// TIA Portal V20 export
FUNCTION_BLOCK "Conveyor_C2"   // FB3, FBD
// stored: Access Published, MemoryReserve 100, Namespace Conveyor2, SetENOAutomatically false
   VAR
      Jog_Right : Bool;
      Jog_Left : Bool;
      Auto_Right : Bool;
      PF_Bay1_NewProd : Bool;
      PF_Bay2_NewProd : Bool;
      PF_Bay3_NewProd : Bool;
      PF_Bay4_EndConv : Bool;
   END_VAR
   VAR_TEMP   // added for the SCL form of the ladder/FBD networks
      _w1 : Bool;
      _w2 : Bool;
      _w3 : Bool;
      _w4 : Bool;
      _w5 : Bool;
      _w6 : Bool;
      _w7 : Bool;
   END_VAR
BEGIN

REGION Network 1: Jog conveyor LEFT
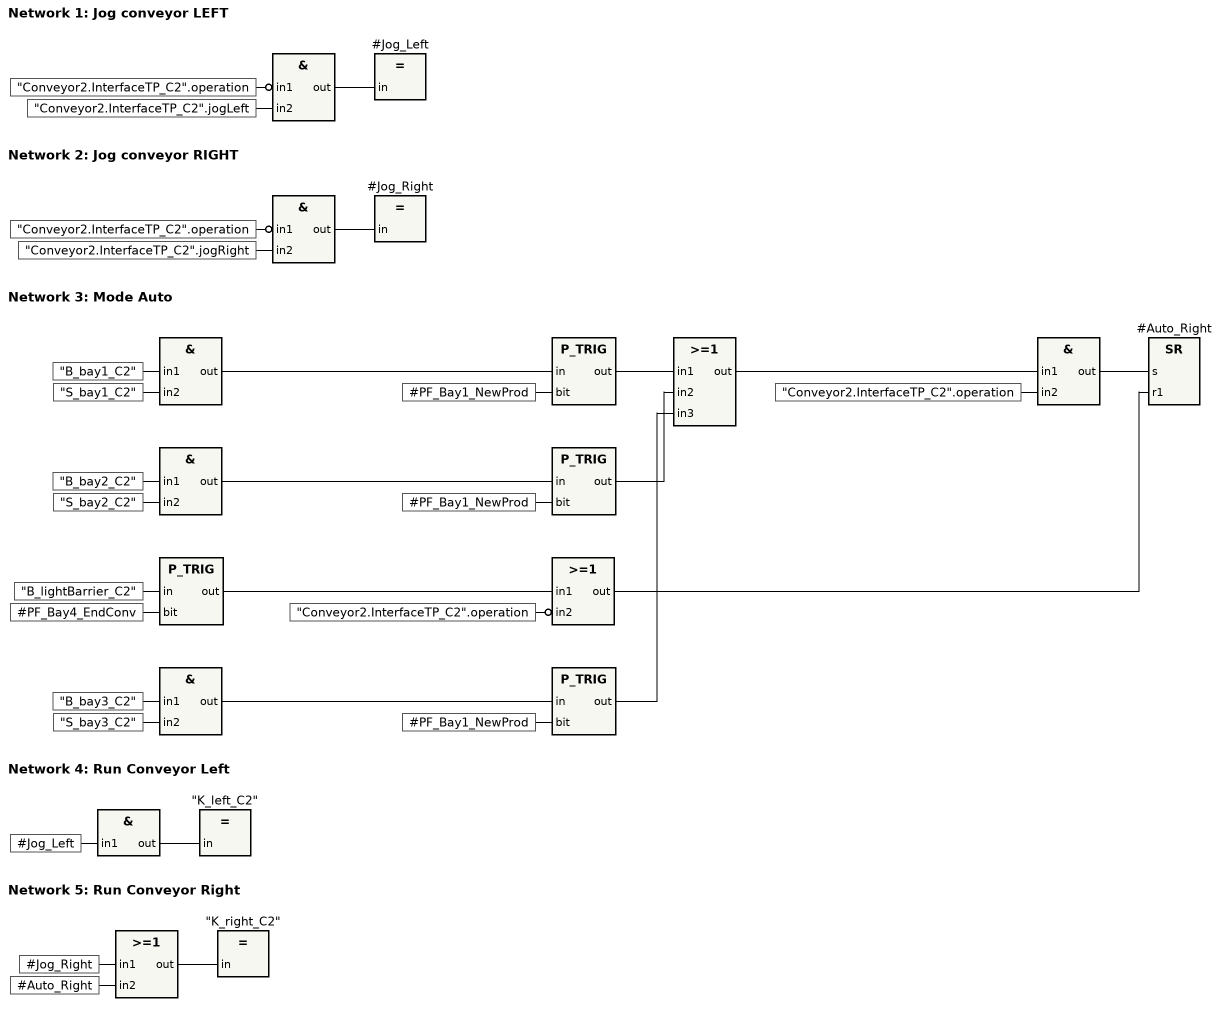
   #Jog_Left := NOT "Conveyor2.InterfaceTP_C2".operation AND "Conveyor2.InterfaceTP_C2".jogLeft;
END_REGION

REGION Network 2: Jog conveyor RIGHT
   #Jog_Right := NOT "Conveyor2.InterfaceTP_C2".operation AND "Conveyor2.InterfaceTP_C2".jogRight;
END_REGION

REGION Network 3: Mode Auto
   // _.K_right_C2
   #_w1 := "B_bay1_C2" AND "S_bay1_C2";
   #_w2 := #_w1 AND NOT #PF_Bay1_NewProd;   // rising edge
   #PF_Bay1_NewProd := #_w1;
   #_w3 := "B_bay2_C2" AND "S_bay2_C2";
   #_w4 := #_w3 AND NOT #PF_Bay1_NewProd;   // rising edge
   #PF_Bay1_NewProd := #_w3;
   #_w5 := "B_bay3_C2" AND "S_bay3_C2";
   #_w6 := #_w5 AND NOT #PF_Bay1_NewProd;   // rising edge
   #PF_Bay1_NewProd := #_w5;
   #_w7 := "B_lightBarrier_C2" AND NOT #PF_Bay4_EndConv;   // rising edge
   #PF_Bay4_EndConv := "B_lightBarrier_C2";
   IF (#_w2 OR #_w4 OR #_w6) AND "Conveyor2.InterfaceTP_C2".operation THEN
       #Auto_Right := TRUE;   // SR flip-flop
   END_IF;
   IF #_w7 OR NOT "Conveyor2.InterfaceTP_C2".operation THEN #Auto_Right := FALSE; END_IF;
END_REGION

REGION Network 4: Run Conveyor Left
   "K_left_C2" := #Jog_Left;
END_REGION

REGION Network 5: Run Conveyor Right
   "K_right_C2" := #Jog_Right OR #Auto_Right;
END_REGION
END_FUNCTION_BLOCK
